// TIA Portal V19 export
FUNCTION "OutputHandler2" : Void   // FC53, STL
{ S7_Optimized_Access := 'TRUE' }
AUTHOR : FLA
FAMILY : UHT
VERSION : 1.0
// Programmer Init: 8953-FLA
// 
// Change Log:
// 
// Date        Change                          Updated by
// ------------------------------------------------------
// 19.04.99    1. Edition                      FLA
// stored: AutoNumber false
BEGIN

NETWORK
TITLE = 
// Item control
// AHV_CLOSED, NO, Ahv barrier closed, with 0 feed-back
      CALL  "Item_Control"
      ( "type"      := 0,  // 0=NO-FB, 1=SET-FB, 2=RES-FB, 3=S/R-FB
        maxTime     := 10,  // Max feed-back MAX_TIME
        itemInfo    := "ItemInfoScada".Items[33],  //AHV_CLOSED
        itemTimer   := "ItemTimerwork".AHV_CLOSED,
        itemStatus  := "ItemStatus".AHV_CLOSED,
        itemCommand := "ItemCommand".AHV_CLOSED,
        resetInput  := "AFI",  // Input for de-energised feed-back
        setInput    := "AFI",  // Input for energised feed-back
        output      := "AHV_CLOSED"  // Output
      );

NETWORK
TITLE = 
// Item control
// AHV_HIGH_LEVEL, NO, Ahv high level, with 0 feed-back
      CALL  "Item_Control"
      ( "type"      := 0,  // 0=NO-FB, 1=SET-FB, 2=RES-FB, 3=S/R-FB
        maxTime     := 10,  // Max feed-back MAX_TIME
        itemInfo    := "ItemInfoScada".Items[34],  //AHV_HIGH_LEVEL
        itemTimer   := "ItemTimerwork".AHV_HIGH_LEVEL,
        itemStatus  := "ItemStatus".AHV_HIGH_LEVEL,
        itemCommand := "ItemCommand".AHV_HIGH_LEVEL,
        resetInput  := "AFI",  // Input for de-energised feed-back
        setInput    := "AFI",  // Input for energised feed-back
        output      := "AHV_HIGH_LEVEL"  // Output
      );


NETWORK
TITLE = 
// Item control
// AHV_READY, NO, Ahv ready, with 0 feed-back
      CALL  "Item_Control"
      ( "type"      := 0,  // 0=NO-FB, 1=SET-FB, 2=RES-FB, 3=S/R-FB
        maxTime     := 10,  // Max feed-back MAX_TIME
        itemInfo    := "ItemInfoScada".Items[35],  //AHV_READY
        itemTimer   := "ItemTimerwork".AHV_READY,
        itemStatus  := "ItemStatus".AHV_READY,
        itemCommand := "ItemCommand".AHV_READY,
        resetInput  := "AFI",  // Input for de-energised feed-back
        setInput    := "AFI",  // Input for energised feed-back
        output      := "AHV_READY"  // Output
      );


NETWORK
TITLE = 
// Item control
// AHV_SHUT_DOWN, NO, Ahv shut down, with 0 feed-back
      CALL  "Item_Control"
      ( "type"      := 0,  // 0=NO-FB, 1=SET-FB, 2=RES-FB, 3=S/R-FB
        maxTime     := 10,  // Max feed-back MAX_TIME
        itemInfo    := "ItemInfoScada".Items[36],  //AHV_SHUT_DOWN
        itemTimer   := "ItemTimerwork".AHV_SHUT_DOWN,
        itemStatus  := "ItemStatus".AHV_SHUT_DOWN,
        itemCommand := "ItemCommand".AHV_SHUT_DOWN,
        resetInput  := "AFI",  // Input for de-energised feed-back
        setInput    := "AFI",  // Input for energised feed-back
        output      := "AHV_SHUT_DOWN"  // Output
      );


NETWORK
TITLE = 
// Item control
// AHV_STERILE, NO, Ahv sterile, with 0 feed-back
      CALL  "Item_Control"
      ( "type"      := 0,  // 0=NO-FB, 1=SET-FB, 2=RES-FB, 3=S/R-FB
        maxTime     := 10,  // Max feed-back MAX_TIME
        itemInfo    := "ItemInfoScada".Items[37],  //AHV_STERILE
        itemTimer   := "ItemTimerwork".AHV_STERILE,
        itemStatus  := "ItemStatus".AHV_STERILE,
        itemCommand := "ItemCommand".AHV_STERILE,
        resetInput  := "AFI",  // Input for de-energised feed-back
        setInput    := "AFI",  // Input for energised feed-back
        output      := "AHV_STERILE"  // Output
      );


NETWORK
TITLE = 
// Item control
// PROD_AVAILABLE, NO, Product available, with 0 feed-back
      CALL  "Item_Control"
      ( "type"      := 0,  // 0=NO-FB, 1=SET-FB, 2=RES-FB, 3=S/R-FB
        maxTime     := 10,  // Max feed-back MAX_TIME
        itemInfo    := "ItemInfoScada".Items[38],  //PROD_AVAILABLE
        itemTimer   := "ItemTimerwork".PROD_AVAILABLE,
        itemStatus  := "ItemStatus".PROD_AVAILABLE,
        itemCommand := "ItemCommand".PROD_AVAILABLE,
        resetInput  := "AFI",  // Input for de-energised feed-back
        setInput    := "AFI",  // Input for energised feed-back
        output      := "PROD_AVAILABLE"  // Output
      );


NETWORK
TITLE = 
// Item control
// RINSE_READY, NO, Rinse ready, with 0 feed-back
      CALL  "Item_Control"
      ( "type"      := 0,  // 0=NO-FB, 1=SET-FB, 2=RES-FB, 3=S/R-FB
        maxTime     := 10,  // Max feed-back MAX_TIME
        itemInfo    := "ItemInfoScada".Items[39],  //RINSE_READY
        itemTimer   := "ItemTimerwork".RINSE_READY,
        itemStatus  := "ItemStatus".RINSE_READY,
        itemCommand := "ItemCommand".RINSE_READY,
        resetInput  := "AFI",  // Input for de-energised feed-back
        setInput    := "AFI",  // Input for energised feed-back
        output      := "RINSE_READY"  // Output
      );


NETWORK
TITLE = 
// Item control
// CAUSTIC_READY, NO, Caustic ready, with 0 feed-back
      CALL  "Item_Control"
      ( "type"      := 0,  // 0=NO-FB, 1=SET-FB, 2=RES-FB, 3=S/R-FB
        maxTime     := 10,  // Max feed-back MAX_TIME
        itemInfo    := "ItemInfoScada".Items[40],  //CAUSTIC_READY
        itemTimer   := "ItemTimerwork".CAUSTIC_READY,
        itemStatus  := "ItemStatus".CAUSTIC_READY,
        itemCommand := "ItemCommand".CAUSTIC_READY,
        resetInput  := "AFI",  // Input for de-energised feed-back
        setInput    := "AFI",  // Input for energised feed-back
        output      := "CAUSTIC_READY"  // Output
      );


NETWORK
TITLE = 
// Item control
// ACID_READY, NO, Acid ready, with 0 feed-back
      CALL  "Item_Control"
      ( "type"      := 0,  // 0=NO-FB, 1=SET-FB, 2=RES-FB, 3=S/R-FB
        maxTime     := 10,  // Max feed-back MAX_TIME
        itemInfo    := "ItemInfoScada".Items[41],  //ACID_READY
        itemTimer   := "ItemTimerwork".ACID_READY,
        itemStatus  := "ItemStatus".ACID_READY,
        itemCommand := "ItemCommand".ACID_READY,
        resetInput  := "AFI",  // Input for de-energised feed-back
        setInput    := "AFI",  // Input for energised feed-back
        output      := "ACID_READY"  // Output
      );


NETWORK
TITLE = 
// Item control
// CIP_FILLER_ENABLE, NO, spare, with 0 feed-back
      CALL  "Item_Control"
      ( "type"      := 0,  // 0=NO-FB, 1=SET-FB, 2=RES-FB, 3=S/R-FB
        maxTime     := 10,  // Max feed-back MAX_TIME
        itemInfo    := "ItemInfoScada".Items[42],  //CIP_FILLER_ENABLE
        itemTimer   := "ItemTimerwork".CIP_FILLER_ENABLE,
        itemStatus  := "ItemStatus".CIP_FILLER_ENABLE,
        itemCommand := "ItemCommand".CIP_FILLER_ENABLE,
        resetInput  := "AFI",  // Input for de-energised feed-back
        setInput    := "AFI",  // Input for energised feed-back
        output      := "CIP_FILLER_ENABLE"  // Output
      );


NETWORK
TITLE = 
// Item control
// Q29_2_NotUsed, , spare, with 0 feed-back
      CALL  "Item_Control"
      ( "type"      := 1,  // 0=NO-FB, 1=SET-FB, 2=RES-FB, 3=S/R-FB
        maxTime     := 10,  // Max feed-back MAX_TIME
        itemInfo    := "ItemInfoScada".Items[43],  //WATER_PUMP
        itemTimer   := "ItemTimerwork".WATER_PUMP,
        itemStatus  := "ItemStatus".WATER_PUMP,
        itemCommand := "ItemCommand".WATER_PUMP,
        resetInput  := "AFI",  // Input for de-energised feed-back
        setInput    := "WaterPumpS",  // Input for energised feed-back
        output      := "WATER_SUPPLY_PUMP"  // Output
      );


NETWORK
TITLE = 
// Item control
// Y0901, NC, valve, with 0 feed-back
      CALL  "Item_Control"
      ( "type"      := 0,  // 0=NO-FB, 1=SET-FB, 2=RES-FB, 3=S/R-FB
        maxTime     := 10,  // Max feed-back MAX_TIME
        itemInfo    := "ItemInfoScada".Items[44],  //Y0901
        itemTimer   := "ItemTimerwork".Y0901,
        itemStatus  := "ItemStatus".Y0901,
        itemCommand := "ItemCommand".Y0901,
        resetInput  := "AFI",  // Input for de-energised feed-back
        setInput    := "AFI",  // Input for energised feed-back
        output      := "Y0901"  // Output
      );


NETWORK
TITLE = 
// Item control
// Y0902, NC, valve, with 0 feed-back
      CALL  "Item_Control"
      ( "type"      := 0,  // 0=NO-FB, 1=SET-FB, 2=RES-FB, 3=S/R-FB
        maxTime     := 10,  // Max feed-back MAX_TIME
        itemInfo    := "ItemInfoScada".Items[45],  //Y0902
        itemTimer   := "ItemTimerwork".Y0902,
        itemStatus  := "ItemStatus".Y0902,
        itemCommand := "ItemCommand".Y0902,
        resetInput  := "AFI",  // Input for de-energised feed-back
        setInput    := "AFI",  // Input for energised feed-back
        output      := "Y0902"  // Output
      );


NETWORK
TITLE = 
// Item control
// Y0903, NC, valve, with 0 feed-back
      CALL  "Item_Control"
      ( "type"      := 0,  // 0=NO-FB, 1=SET-FB, 2=RES-FB, 3=S/R-FB
        maxTime     := 10,  // Max feed-back MAX_TIME
        itemInfo    := "ItemInfoScada".Items[46],  //Y0903
        itemTimer   := "ItemTimerwork".Y0903,
        itemStatus  := "ItemStatus".Y0903,
        itemCommand := "ItemCommand".Y0903,
        resetInput  := "AFI",  // Input for de-energised feed-back
        setInput    := "AFI",  // Input for energised feed-back
        output      := "Y0903"  // Output
      );


NETWORK
TITLE = 
// Item control
// TANK_READY, NO, Signal to uht tank ready, with 0 feed-back
      CALL  "Item_Control"
      ( "type"      := 0,  // 0=NO-FB, 1=SET-FB, 2=RES-FB, 3=S/R-FB
        maxTime     := 10,  // Max feed-back MAX_TIME
        itemInfo    := "ItemInfoScada".Items[47],  //TANK_READY
        itemTimer   := "ItemTimerwork".TANK_READY,
        itemStatus  := "ItemStatus".TANK_READY,
        itemCommand := "ItemCommand".TANK_READY,
        resetInput  := "AFI",  // Input for de-energised feed-back
        setInput    := "AFI",  // Input for energised feed-back
        output      := "TANK_READY"  // Output
      );


NETWORK
TITLE = 
// Item control
// TANK_OPEN, NO, Signal to uht tank open, with 0 feed-back
      CALL  "Item_Control"
      ( "type"      := 0,  // 0=NO-FB, 1=SET-FB, 2=RES-FB, 3=S/R-FB
        maxTime     := 10,  // Max feed-back MAX_TIME
        itemInfo    := "ItemInfoScada".Items[48],  //TANK_OPEN
        itemTimer   := "ItemTimerwork".TANK_OPEN,
        itemStatus  := "ItemStatus".TANK_OPEN,
        itemCommand := "ItemCommand".TANK_OPEN,
        resetInput  := "AFI",  // Input for de-energised feed-back
        setInput    := "AFI",  // Input for energised feed-back
        output      := "TANK_OPEN"  // Output
      );


NETWORK
TITLE = 
// Item control
// Y0904, NC, valve, with 2 feed-back
      CALL  "Item_Control"
      ( "type"      := 3,  // 0=NO-FB, 1=SET-FB, 2=RES-FB, 3=S/R-FB
        maxTime     := 10,  // Max feed-back MAX_TIME
        itemInfo    := "ItemInfoScada".Items[49],  //Y0904
        itemTimer   := "ItemTimerwork".Y0904,
        itemStatus  := "ItemStatus".Y0904,
        itemCommand := "ItemCommand".Y0904,
        resetInput  := "Y0904R",  // Input for de-energised feed-back
        setInput    := "Y0904S",  // Input for energised feed-back
        output      := "Y0904"  // Output
      );

NETWORK
TITLE = 
// Item control
// Y0905, NC, valve, with 2 feed-back
      CALL  "Item_Control"
      ( "type"      := 3,  // 0=NO-FB, 1=SET-FB, 2=RES-FB, 3=S/R-FB
        maxTime     := 10,  // Max feed-back MAX_TIME
        itemInfo    := "ItemInfoScada".Items[50],  //Y0905
        itemTimer   := "ItemTimerwork".Y0905,
        itemStatus  := "ItemStatus".Y0905,
        itemCommand := "ItemCommand".Y0905,
        resetInput  := "Y0905R",  // Input for de-energised feed-back
        setInput    := "Y0905S",  // Input for energised feed-back
        output      := "Y0905"  // Output
      );


NETWORK
TITLE = 
// Item control
// Y0906, NC, valve, with 2 feed-back
      CALL  "Item_Control"
      ( "type"      := 3,  // 0=NO-FB, 1=SET-FB, 2=RES-FB, 3=S/R-FB
        maxTime     := 10,  // Max feed-back MAX_TIME
        itemInfo    := "ItemInfoScada".Items[51],  //Y0906
        itemTimer   := "ItemTimerwork".Y0906,
        itemStatus  := "ItemStatus".Y0906,
        itemCommand := "ItemCommand".Y0906,
        resetInput  := "Y0906R",  // Input for de-energised feed-back
        setInput    := "Y0906S",  // Input for energised feed-back
        output      := "Y0906"  // Output
      );


NETWORK
TITLE = 
// Item control
// Y0907, NC, valve, with 2 feed-back
      CALL  "Item_Control"
      ( "type"      := 3,  // 0=NO-FB, 1=SET-FB, 2=RES-FB, 3=S/R-FB
        maxTime     := 10,  // Max feed-back MAX_TIME
        itemInfo    := "ItemInfoScada".Items[52],  //Y0907
        itemTimer   := "ItemTimerwork".Y0907,
        itemStatus  := "ItemStatus".Y0907,
        itemCommand := "ItemCommand".Y0907,
        resetInput  := "Y0907R",  // Input for de-energised feed-back
        setInput    := "Y0907S",  // Input for energised feed-back
        output      := "Y0907"  // Output
      );


NETWORK
TITLE = 
// Item control
// Y0908, NC, valve, with 2 feed-back
      CALL  "Item_Control"
      ( "type"      := 3,  // 0=NO-FB, 1=SET-FB, 2=RES-FB, 3=S/R-FB
        maxTime     := 10,  // Max feed-back MAX_TIME
        itemInfo    := "ItemInfoScada".Items[53],  //Y0908
        itemTimer   := "ItemTimerwork".Y0908,
        itemStatus  := "ItemStatus".Y0908,
        itemCommand := "ItemCommand".Y0908,
        resetInput  := "Y0908R",  // Input for de-energised feed-back
        setInput    := "Y0908S",  // Input for energised feed-back
        output      := "Y0908"  // Output
      );


NETWORK
TITLE = 
// Item control
// Y0909, NC, valve, with 2 feed-back
      CALL  "Item_Control"
      ( "type"      := 3,  // 0=NO-FB, 1=SET-FB, 2=RES-FB, 3=S/R-FB
        maxTime     := 10,  // Max feed-back MAX_TIME
        itemInfo    := "ItemInfoScada".Items[54],  //Y0909
        itemTimer   := "ItemTimerwork".Y0909,
        itemStatus  := "ItemStatus".Y0909,
        itemCommand := "ItemCommand".Y0909,
        resetInput  := "Y0909R",  // Input for de-energised feed-back
        setInput    := "Y0909S",  // Input for energised feed-back
        output      := "Y0909"  // Output
      );


NETWORK
TITLE = 
// Item control
// Y0910, NC, valve, with 2 feed-back
      CALL  "Item_Control"
      ( "type"      := 3,  // 0=NO-FB, 1=SET-FB, 2=RES-FB, 3=S/R-FB
        maxTime     := 10,  // Max feed-back MAX_TIME
        itemInfo    := "ItemInfoScada".Items[55],  //Y0910
        itemTimer   := "ItemTimerwork".Y0910,
        itemStatus  := "ItemStatus".Y0910,
        itemCommand := "ItemCommand".Y0910,
        resetInput  := "Y0910R",  // Input for de-energised feed-back
        setInput    := "Y0910S",  // Input for energised feed-back
        output      := "Y0910"  // Output
      );


NETWORK
TITLE = 
// Item control
// Y0911, NC, valve, with 2 feed-back
      CALL  "Item_Control"
      ( "type"      := 3,  // 0=NO-FB, 1=SET-FB, 2=RES-FB, 3=S/R-FB
        maxTime     := 10,  // Max feed-back MAX_TIME
        itemInfo    := "ItemInfoScada".Items[56],  //Y0911
        itemTimer   := "ItemTimerwork".Y0911,
        itemStatus  := "ItemStatus".Y0911,
        itemCommand := "ItemCommand".Y0911,
        resetInput  := "Y0911R",  // Input for de-energised feed-back
        setInput    := "Y0911S",  // Input for energised feed-back
        output      := "Y0911"  // Output
      );


NETWORK
TITLE = 
// Item control
// Y0912, NC, valve, with 2 feed-back
      CALL  "Item_Control"
      ( "type"      := 3,  // 0=NO-FB, 1=SET-FB, 2=RES-FB, 3=S/R-FB
        maxTime     := 10,  // Max feed-back MAX_TIME
        itemInfo    := "ItemInfoScada".Items[57],  //Y0912
        itemTimer   := "ItemTimerwork".Y0912,
        itemStatus  := "ItemStatus".Y0912,
        itemCommand := "ItemCommand".Y0912,
        resetInput  := "Y0912R",  // Input for de-energised feed-back
        setInput    := "Y0912S",  // Input for energised feed-back
        output      := "Y0912"  // Output
      );


NETWORK
TITLE = 
// Item control
// Q41_1_NotUsed, , spare, with 0 feed-back
      CALL  "Item_Control"
      ( "type"      := 0,  // 0=NO-FB, 1=SET-FB, 2=RES-FB, 3=S/R-FB
        maxTime     := 10,  // Max feed-back MAX_TIME
        itemInfo    := "ItemInfoScada".Items[58],  //Q41_1
        itemTimer   := "ItemTimerwork".Q41_1,
        itemStatus  := "ItemStatus".Q41_1,
        itemCommand := "ItemCommand".Q41_1,
        resetInput  := "AFI",  // Input for de-energised feed-back
        setInput    := "AFI",  // Input for energised feed-back
        output      := "steam_lp_enabled"  // Output
      );

NETWORK
TITLE = 
// Item control
// CIP_Route, , spare, with 0 feed-back
      CALL  "Item_Control"
      ( "type"      := 0,  // 0=NO-FB, 1=SET-FB, 2=RES-FB, 3=S/R-FB
        maxTime     := 10,  // Max feed-back MAX_TIME
        itemInfo    := "ItemInfoScada".Items[59],  //CIP_Route
        itemTimer   := "ItemTimerwork".CIP_Route,
        itemStatus  := "ItemStatus".CIP_Route,
        itemCommand := "ItemCommand".CIP_Route,
        resetInput  := "AFI",  // Input for de-energised feed-back
        setInput    := "AFI",  // Input for energised feed-back
        output      := "CIP_Route"  // Output
      );


NETWORK
TITLE = 
// Item control
// Sterilisation_Steam, , spare, with 0 feed-back
      CALL  "Item_Control"
      ( "type"      := 0,  // 0=NO-FB, 1=SET-FB, 2=RES-FB, 3=S/R-FB
        maxTime     := 10,  // Max feed-back MAX_TIME
        itemInfo    := "ItemInfoScada".Items[60],  //SIP_Steam
        itemTimer   := "ItemTimerwork".SIP_Steam,
        itemStatus  := "ItemStatus".SIP_Steam,
        itemCommand := "ItemCommand".SIP_Steam,
        resetInput  := "AFI",  // Input for de-energised feed-back
        setInput    := "AFI",  // Input for energised feed-back
        output      := "Sterilisation_Steam"  // Output
      );


NETWORK
TITLE = 
// Item control
// Product_Available, , spare, with 0 feed-back
      CALL  "Item_Control"
      ( "type"      := 0,  // 0=NO-FB, 1=SET-FB, 2=RES-FB, 3=S/R-FB
        maxTime     := 10,  // Max feed-back MAX_TIME
        itemInfo    := "ItemInfoScada".Items[61],  //PROD_AVAILABLE
        itemTimer   := "ItemTimerwork".PROD_AVAILABLE,
        itemStatus  := "ItemStatus".PROD_AVAILABLE,
        itemCommand := "ItemCommand".PROD_AVAILABLE,
        resetInput  := "AFI",  // Input for de-energised feed-back
        setInput    := "AFI",  // Input for energised feed-back
        output      := "Product_Available"  // Output
      );


NETWORK
TITLE = 
// Item control
// Barrier_Sterile, , spare, with 0 feed-back
      CALL  "Item_Control"
      ( "type"      := 0,  // 0=NO-FB, 1=SET-FB, 2=RES-FB, 3=S/R-FB
        maxTime     := 10,  // Max feed-back MAX_TIME
        itemInfo    := "ItemInfoScada".Items[62],  //Barrier_Sterile
        itemTimer   := "ItemTimerwork".Barrier_Sterile,
        itemStatus  := "ItemStatus".Barrier_Sterile,
        itemCommand := "ItemCommand".Barrier_Sterile,
        resetInput  := "AFI",  // Input for de-energised feed-back
        setInput    := "AFI",  // Input for energised feed-back
        output      := "Barrier_Sterile"  // Output
      );


NETWORK
TITLE = 
// Item control
// Product_Route, , spare, with 0 feed-back
      CALL  "Item_Control"
      ( "type"      := 0,  // 0=NO-FB, 1=SET-FB, 2=RES-FB, 3=S/R-FB
        maxTime     := 10,  // Max feed-back MAX_TIME
        itemInfo    := "ItemInfoScada".Items[63],  //Product_Route
        itemTimer   := "ItemTimerwork".Product_Route,
        itemStatus  := "ItemStatus".Product_Route,
        itemCommand := "ItemCommand".Product_Route,
        resetInput  := "AFI",  // Input for de-energised feed-back
        setInput    := "AFI",  // Input for energised feed-back
        output      := "Product_Route"  // Output
      );


NETWORK
TITLE = 
// Item control
// X0913, NC, lamp, with 0 feed-back
      CALL  "Item_Control"
      ( "type"      := 0,  // 0=NO-FB, 1=SET-FB, 2=RES-FB, 3=S/R-FB
        maxTime     := 10,  // Max feed-back MAX_TIME
        itemInfo    := "ItemInfoScada".Items[64],  //X0913
        itemTimer   := "ItemTimerwork".X0913,
        itemStatus  := "ItemStatus".X0913,
        itemCommand := "ItemCommand".X0913,
        resetInput  := "AFI",  // Input for de-energised feed-back
        setInput    := "AFI",  // Input for energised feed-back
        output      := "X0913"  // Output
      );

END_FUNCTION
